FUNCTION_BLOCK PUBLIC FB_EL6001_RS232
VAR_IN_OUT
	LineCtrl : FB_EL6001_LINE_CTRL;
END_VAR
VAR_INPUT
	Send : BOOL;
END_VAR
VAR_OUTPUT
END_VAR
VAR
	ReceiveString : ReceiveString255;
	SendString : SendString255;
	RecvStr : STRING[255];
	SendStr : STRING[255];
END_VAR

ReceiveString(RXbuffer := LineCtrl.RxBuffer, ReceivedString := RecvStr, Timeout := T#1S);

IF Send THEN
	SendString(TXbuffer := LineCtrl.TxBuffer, SendString := SendStr);
	IF NOT SendString.Busy THEN
		Send := FALSE;
	END_IF;
END_IF;

END_FUNCTION_BLOCK

(* stored: Version 1.1.0.1, ProductVersion 3.1.4024.12
   POU FB_EL6001_RS232: Id {e3559a5b-0108-4532-aafa-a35846972476}, SpecialFunc None *)
